(*
Represents a receiver in the Broadcast system. Implements the necessary methods for receiving events and pairing signals.
*)
FUNCTION_BLOCK FINAL Receiver IMPLEMENTS I_ReceiverNode, I_Receiver
VAR
	
	_comp			: Component(THIS^);
	_tag			: TagBase;
	_iCallable		: I_Callable;
	_bIsOk			: BOOL := TRUE;
END_VAR

//FB_Init is always available implicitly and it is used primarily for initialization.
//The return value is not evaluated. For a specific influence, you can also declare the
//methods explicitly and provide additional code there with the standard initialization
//code. You can evaluate the return value.
METHOD FB_Init: BOOL
VAR_INPUT
    bInitRetains: BOOL; // TRUE: the retain variables are initialized (reset warm / reset cold)
    bInCopyCode: BOOL;  // TRUE: the instance will be copied to the copy code afterward (online change)

	iCallable	: I_Callable;
END_VAR
_iCallable := iCallable;
IF _iCallable = 0 THEN
	_bIsOk := FALSE;
	DebugMsg(THIS^, 'iReceiver = 0!');
END_IF
END_METHOD

(*
Checks if the receiver is properly initialized and ready to operate.
*)
PROPERTY INTERNAL IsOk : BOOL
GET
IsOk := _bIsOk;
END_GET
END_PROPERTY

(*
Pairs the receiver with a signal.  
Returns:
- `Ok` - If pairing is successful.
- `Err.Itf0` - If the receiver interface is invalid.
- `Err.IncArg` - If the `I_Receiver` is invalid.
- `Err.ItfEq` - If the `I_Receiver` is already paired with this `I_Signal`.
- `Err.Ovf` - If there is no space for another pairing.
*)
METHOD Pair : Result
VAR_INPUT
	iSignal		: I_Signal;
END_VAR
IF iSignal <> 0 THEN
	Pair := iSignal.Pair(THIS^);
ELSE
	Pair := Error;
END_IF
END_METHOD

METHOD INTERNAL Receive
VAR_INPUT
	iArg			: I_Arg;
END_VAR
_iCallable.Call(iArg);
END_METHOD

(*
Provides access to the tag associated with the signal.
*)
PROPERTY Tag : I_Tag
GET
Tag := _tag;
END_GET
END_PROPERTY

(*
Unpairs the signal from a specified receiver.
Returns:
- `Ok` - If unpairing is successful.
- `Err.Itf0` - If the receiver interface is invalid.
- `Err.IncArg` - If the `I_Receiver` is invalid.
- `Err.NoMatch` - If `I_Signal` is not paired with this `I_Receiver`.
*)
METHOD Unpair : Result
VAR_INPUT
	iSignal		: I_Signal;
END_VAR
IF iSignal <> 0 THEN
	Unpair := iSignal.Unpair(THIS^);
ELSE
	Unpair := Error;
END_IF
END_METHOD

END_FUNCTION_BLOCK

(* stored: Version 1.1.0.1
   POU Receiver: Id {09249f88-9a26-4648-82ad-ef06a2e8297b}, SpecialFunc None
   Method FB_init: Id {180c7f71-8e66-475d-822f-48b13e0266b6}
   Property IsOk: Id {f1f087c9-ce24-4a7a-9d2f-520cd51dc062}
   Get Get: Id {01cfd46c-ea36-47ad-88cc-581ac680254f}
   Method Pair: Id {6fffc843-9230-4d39-885d-576d2d6aa59f}
   Method Receive: Id {7cf97b80-2026-43ed-bd4a-a4b08dba024b}
   Property Tag: Id {c4ff52e5-e8db-4834-b8d3-e55ed4dc8f91}
   Get Get: Id {78444fd4-17bd-40e5-bca6-e460c617c742}
   Method Unpair: Id {9cdd6e18-8337-45bf-81f7-8c24c8d9cdfa} *)
